INTERFACE ITF_Group3_HMI_Connector_Command EXTENDS ITF_BaseGroupElement_HMI_Connector_Command

END_INTERFACE

(* stored: Version 1.1.0.1
   Itf ITF_Group3_HMI_Connector_Command: Id {a380b94d-a37b-0a8d-288e-6b6697890885} *)
